(*

.. <legal notes>

legal notes
=================
| SPDX-FileCopyrightText: © 2026 Oleksandr Tiutyk <trofimich@gmail.com>
| SPDX-License-Identifier: LGPL-3.0-only
| For details check: LGPL-3.0-only_

.. _LGPL-3.0-only: https://www.gnu.org/licenses/lgpl-3.0.en.html

.. </legal notes>

*)

INTERFACE IDevice EXTENDS IChildAutomationComponent

METHOD Initialize : BOOL
END_METHOD

END_INTERFACE

(* stored: Version 1.1.0.1
   Itf IDevice: Id {9736df80-aba4-4bb1-a085-478863d519b5}
   Method Initialize: Id {c1b642e1-c838-4d11-be0f-d347cee28d0c} *)
